// TIA Portal project "simzamanlama" (V16)

(* hardware
DEVICE "S71500/ET200MP station_1"  S7-1500 station
   slot 0: "Rail_0"  Rack  6ES7 590-1***0-0AA0
   slot 1: "PLC_1"  CPU 1511C-1 PN  6ES7 511-1CK00-0AB0  V2.8
      slot 3: "CPU display_1"  6ES7591-1AA00-0AA0
      slot 32768: "PROFINET interface_1"  X1
         slot 32769: "Port_1"  X1 P1
         slot 32770: "Port_2"  X1 P2
      slot 34817: "Virtual CP interface port_1"  Virtual CP interface port  Virtual CP interface port
*)

// ===== PLC "PLC_1"  CPU 1511C-1 PN =====

VAR_GLOBAL   // PLC tag table "Default tag table"
   ""start"" AT %I0.0 : Bool;
   ""stop"" AT %I0.1 : Bool;
   ""motor1"" AT %Q0.1 : Bool;
   ""motor2"" AT %Q0.2 : Bool;
   ""motor3"" AT %Q0.3 : Bool;
END_VAR